{attribute 'qualified_only'}
{attribute 'strict'}
TYPE act_type :
(
	linear := 0,
	relu :=1,
	tanh :=2,
	normalization := 10,
	denormalization :=11
);
END_TYPE

(* stored: Version 1.1.0.1, ProductVersion 3.1.4024.12
   DUT act_type: Id {a4894a0e-41f6-414c-9a45-a6a9800ade25} *)
